PROGRAM MAIN
VAR
	fbGetHostname : FB_GetHostName;
END_VAR

PRG_READ(); // Call sample for UA_Read
//PRG_READ_IndexRange(); // Call sample for UA_Read
//PRG_READ_List(); // Call sample for UA_ReadList
//PRG_READ_List_Array(); // Call sample for UA_ReadList to read array elements
//PRG_WRITE(); // Call sample for UA_Write
//PRG_WRITE_IndexRange(); // Call sample for UA_Write
//PRG_METHOD(); // Call sample for UA_MethodCall

END_PROGRAM

(* stored: Version 1.1.0.1, ProductVersion 3.1.4024.3
   POU MAIN: Id {fc8ad144-f214-4b14-b487-cf23eecee195}, SpecialFunc None *)
